PROGRAM MAIN
VAR
	bChange : BOOL := TRUE;
	bAnother : BOOL := FALSE;
	FinalTest1 : FB_FinalTest;
END_VAR

IF bChange THEN
	FinalTest1();
END_IF

END_PROGRAM

(* stored: Version 1.1.0.1, ProductVersion 3.1.4024.9
   POU MAIN: Id {3e384c1b-24f7-4744-81bf-b6f9c0d42fbb}, SpecialFunc None *)
